// TIA Portal V16 export
// export: Created 2023-03-29T11:03:45.7704022Z, ExportSetting WithDefaults, DisplayName Totally Integrated Automation Portal, DisplayVersion V16 Update 6, DisplayName TIA Portal Version Control Interface, DisplayVersion V16 Update 2, DisplayName TIA Portal Openness, DisplayVersion V16 Update 6, DisplayName STEP 7 Professional, DisplayVersion V16 Update 6, DisplayName STEP 7 Safety, DisplayVersion V16, DisplayName WinCC Advanced, DisplayVersion V16 Update 6
VAR_GLOBAL   // PLC tag table "Z10"
   inputOtwartaZ_10 AT %M72.2 : Bool;   // znacznik wejście
   Hbit_Otwórz_Z10 AT %M28.4 : Bool;
   Hbit_Auto_Manu_Z10 AT %M28.7 : Bool;
   setSVMC_Z_10 AT %M73.3 : Bool;   // Znacznik polecenia zamknij w trybie automat
   setSVMO_Z_10 AT %M73.2 : Bool;   // Znacznik polecenia otwórz w trybie automat
   Hbit_Zamknieta_Z10 AT %M28.3 : Bool;
   setAlarm_Moment_Z_10 AT %M73.4 : Bool;   // znacznik alarmu od momentówki w trybie zdalnym (aut/mamnual)
   inputAumaautomatZ_10 AT %M72.7 : Bool;   // znacznik wejście
   CMD_Close_Z_10 AT %M73.6 : Bool;   // załącz zamykanie
   CMD_Open_Z_10 AT %M73.5 : Bool;   // załącz otwieranie
   inputRuch_Z_10 AT %M72.4 : Bool;   // znacznik wejście
   Byte_Status_Z10 AT %MW28 : Word;   // Słowo statusu napędu
   inputREMT_Z_10 AT %M72.1 : Bool;   // znacznik wejście zdalne
   Hbit_REN_Z10 AT %M28.2 : Bool;
   Hbit_Otwarta_Z10 AT %M28.1 : Bool;
   Hbit_Reset_Z10 AT %M28.6 : Bool;
   inputAumaawariaZ_10 AT %M73.1 : Bool;   // znacznik wejście
   inputAumagotowośćZ_10 AT %M73.0 : Bool;   // znacznik wejście
   Hbit_Zamknij_Z10 AT %M28.5 : Bool;
   CMD_Awaria_Z_10 AT %M73.7 : Bool;   // Awaria zbiorcza
   inputAumalokalneZ_10 AT %M72.6 : Bool;   // znacznik wejście
   isGotowość_Z_10 AT %M72.0 : Bool;   // bit gotowości wspólny
   inputZamkniętaZ_10 AT %M72.3 : Bool;   // znacznik wejście
   Hbit_Alarm_Z10 AT %M28.0 : Bool;
   isOpen_Z10 AT %M52.3 : Bool;   // bit potwierdzenia otwarcia prz sterowaniu [%]
   inputAwariaMomentZ_10 AT %M72.5 : Bool;   // znacznik wejście
   isClose_od_położenia AT %M74.0 : Bool;   // gdy brak sygnały a krancowego wyłacznika to patrzy na pozycję z nadajnika
END_VAR
